(* CODESYS project Initial_Program.project
   Version: 0.0.0.0
   Title: Initial_Program
   Author: MYBOOK

Project tree, tasks and I/O mapping:
  Skripsi_Yosef : TM262L10MESE8T, Schneider Electric, order no. TM262L10MESE8T, version 5.0.4.83
      settings: Enable OPC-UA Server = True; BinaryFileSize = 1168; Dhcps Host 0.Client Device Name = 'DEVICE_1'; Dhcps Host 0.Client IP Address = [192, 168, 3, 200]; Dhcps Host 0.Network Mask = [255, 255, 255, 0]; Dhcps Host 0.Default Gateway = [192, 168, 3, 254]; Dhcps Host 1.Client Device Name = 'DEVICE_2'; Dhcps Host 1.Client IP Address = [192, 168, 3, 100]; Dhcps Host 1.Network Mask = [255, 255, 255, 0]; Dhcps Host 1.Default Gateway = [192, 168, 3, 254]; Dhcps Host 2.Client Device Name = 'DEVICE_3'; Dhcps Host 2.Client IP Address = [192, 168, 3, 201]; Dhcps Host 2.Network Mask = [255, 255, 255, 0]; Dhcps Host 2.Default Gateway = [192, 168, 3, 254]; Dhcps Host 3.Client Device Name = 'DEVICE_4'; Dhcps Host 3.Client IP Address = [192, 168, 3, 101]; Dhcps Host 3.Network Mask = [255, 255, 255, 0]; Dhcps Host 3.Default Gateway = [192, 168, 3, 254]; Dhcps Host 4.Client Device Name = 'DEVICE_5'; Dhcps Host 4.Client IP Address = [192, 168, 3, 203]; Dhcps Host 4.Network Mask = [255, 255, 255, 0]; Dhcps Host 4.Default Gateway = [192, 168, 3, 254]; Dhcps Host 5.Client Device Name = 'DEVICE_6'; Dhcps Host 5.Client IP Address = [192, 168, 3, 202]; Dhcps Host 5.Network Mask = [255, 255, 255, 0]; Dhcps Host 5.Default Gateway = [192, 168, 3, 254]; InterfaceUsedByDhcpSize = 4; InterfaceUsedByDhcp = [192,168,3,254]
    application Application
      task MAST (cyclic, interval 10 ms, priority 15, watchdog 50 ms x 1) calls SR_Main
      program SR_Main [LD]
      global variables GVL
      program POU [SFC]
    Machine Assistant
    Message Logger
    COM_Bus : COM Bus - TMS, Schneider Electric, version 5.0.4.83
    Ethernet_1 : ETH1, Schneider Electric, version 5.0.4.83
        settings: DeviceName = 'M262'; WebServer = FALSE; FTP Server = TRUE; SoMachine Protocol = FALSE; Modbus Server = FALSE; NetManage Protocol = FALSE; SNMP protocol = FALSE; WebVisu protocol = FALSE; DHCP Server Active = TRUE; Secured Web Server = TRUE; Remote Connection = FALSE
    Ethernet_2 : ETH2, Schneider Electric, version 5.0.4.83
        settings: IPAddress = [192, 168, 3, 254]; SubnetMask = [255, 255, 255, 0]; GatewayAddress = [192, 168, 3, 1]; DeviceName = 'M262_PLC'; WebServer = TRUE; FTP Server = FALSE; SoMachine Protocol = TRUE; Modbus Server = TRUE; NetManage Protocol = TRUE; SNMP protocol = TRUE; WebVisu protocol = TRUE; DHCP Server Active = TRUE; Secured Web Server = TRUE; Remote Connection = TRUE
      Modbus_TCP_IO_Scanner : Modbus TCP IO Scanner, Schneider Electric, version 1.0.0.12
          unmapped channels: Global Status, Healthbit 0, Healthbit 1, Healthbit 2, Healthbit 3
        OT_Sensor_Temp_Humid : Generic Modbus TCP Slave, Schneider Electric, version 1.0.2.21
            settings: DeviceNumber = 512; Object Input1 = [128, 2, 21233664, 0]; Unit-ID = 248; IPAddress = [192, 168, 3, 200]; GatewayAddress = [192, 168, 3, 254]; DeviceName = 'DEVICE_1'; Channel 0.Channel ID = 0; Channel 0.Unit-ID = 1; Channel 0.Repetition Rate = 100; Channel 0.Function Code = 3; Channel 0.Read Offset = 16#0000; Channel 0.Read Length = 2; Channel 0.Write Offset = 0; Channel 0.Write Length = 0
            unmapped channels: Channel 0, Channel 0
        AHU_Act_Remote_AC : Generic Modbus TCP Slave, Schneider Electric, version 1.0.2.21
            settings: DeviceNumber = 513; Object Output1 = [131, 2, 25428068, 1]; Unit-ID = 248; IPAddress = [192, 168, 3, 100]; GatewayAddress = [192, 168, 3, 254]; DeviceName = 'DEVICE_2'; Channel 1.Channel ID = 1; Channel 1.Unit-ID = 255; Channel 1.Repetition Rate = 100; Channel 1.Function Code = 16; Channel 1.Read Offset = 0; Channel 1.Read Length = 0; Channel 1.Write Offset = 16#0064; Channel 1.Write Length = 2
            unmapped channels: Channel 1, Channel 1
        OT_Sensor_Press_Temp : Generic Modbus TCP Slave, Schneider Electric, version 1.0.2.21
            settings: DeviceNumber = 514; Object Input1 = [132, 2, 21233764, 2]; Unit-ID = 248; IPAddress = [192, 168, 3, 201]; GatewayAddress = [192, 168, 3, 254]; DeviceName = 'DEVICE_3'; Channel 1.Channel ID = 2; Channel 1.Unit-ID = 255; Channel 1.Repetition Rate = 100; Channel 1.Function Code = 3; Channel 1.Read Offset = 16#0064; Channel 1.Read Length = 2; Channel 1.Write Offset = 0; Channel 1.Write Length = 0
            unmapped channels: Channel 1, Channel 1
        AHU_Act_Motor_Exhaust : Generic Modbus TCP Slave, Schneider Electric, version 1.0.2.21
            settings: DeviceNumber = 515; Object Output1 = [135, 8, 25427968, 3]; Unit-ID = 248; IPAddress = [192, 168, 3, 101]; GatewayAddress = [192, 168, 3, 254]; DeviceName = 'DEVICE_4'; Channel 3.Channel ID = 3; Channel 3.Unit-ID = 1; Channel 3.Repetition Rate = 100; Channel 3.Function Code = 16; Channel 3.Read Offset = 0; Channel 3.Read Length = 0; Channel 3.Write Offset = 16#0000; Channel 3.Write Length = 8
            unmapped channels: Channel 3, Channel 3, Channel 3, Channel 3, Channel 3, Channel 3, Channel 3, Channel 3
        AHU_Sensor_Temp_Humid_Pressure : Generic Modbus TCP Slave, Schneider Electric, version 1.0.2.21
            settings: DeviceNumber = 516; Object Input1 = [136, 4, 21233764, 4]; Unit-ID = 248; IPAddress = [192, 168, 3, 203]; GatewayAddress = [192, 168, 3, 254]; DeviceName = 'DEVICE_5'; Channel 4.Channel ID = 4; Channel 4.Unit-ID = 255; Channel 4.Repetition Rate = 20; Channel 4.Function Code = 3; Channel 4.Read Offset = 16#0064; Channel 4.Read Length = 4; Channel 4.Write Offset = 0; Channel 4.Write Length = 0
            unmapped channels: Channel 4, Channel 4, Channel 4, Channel 4
        Outdoor_Sensor_Press_temp : Generic Modbus TCP Slave, Schneider Electric, version 1.0.2.21
            settings: DeviceNumber = 517; Object Input1 = [138, 2, 21233764, 5]; Unit-ID = 248; IPAddress = [192, 168, 3, 202]; GatewayAddress = [192, 168, 3, 254]; DeviceName = 'DEVICE_6'; Channel 5.Channel ID = 5; Channel 5.Unit-ID = 255; Channel 5.Repetition Rate = 20; Channel 5.Function Code = 3; Channel 5.Read Offset = 16#0064; Channel 5.Read Length = 2; Channel 5.Write Offset = 0; Channel 5.Write Length = 0
            unmapped channels: Channel 5, Channel 5
    Serial_Line : Serial line, Schneider Electric, version 5.0.4.83
      Machine_Expert_Network_Manager : Machine Expert-Network Manager, Schneider Electric, version 4.0.0.3
    DI : Digital Inputs, Schneider Electric, version 5.0.4.83
        input  ibDI_IB0 : BYTE  // IB0
        input  ibDI_IB1 : BYTE  // IB1
    DQ : Digital Outputs, Schneider Electric, version 5.0.4.83
        unmapped channels: QB0, QB1
    IO_Bus : IO bus - TM3, Schneider Electric, version 5.0.4.83
  FdtConnections : FDT Connections, Schneider Electric, version 1.0.0.2
  Project Information/
    function GetCompany [ST]
    function GetTitle [ST]
    function GetVersion [ST]
    function GetTextProperty [ST]
    function GetTextProperty2 [ST]
    function GetNumberProperty [ST]
    function GetBooleanProperty [ST]
    function GetVersionProperty [ST]
*)

// Skripsi_Yosef/Application/GVL
{attribute 'qualified_only'}
VAR_GLOBAL
	
END_VAR

// Skripsi_Yosef/Application/SR_Main
PROGRAM SR_Main
VAR
	AC_StatusHMI AT %MX6.0: BOOL := FALSE;
	OT_Temp AT %MW0: WORD;
	OT_Humid AT %MW1: WORD;
	OT_Pressure AT %MW2: WORD;
	AC_Status AT %MW4: WORD;
	AC_Temp AT %MW5: WORD := 24;
	AC_TempUp AT %MX12.0: BOOL;
	AC_TempDown AT %MX12.1: BOOL;
	AC_TempRST AT %MX12.2: BOOL;
	AHU_Temp AT %MW7: WORD;
	AHU_Humid AT %MW8: WORD;
	AHU_Press AT %MW9: WORD;
	AHU_FanOverride AT %MX20.0: BOOL;
	HMI_FANSpeed1 AT %MW11: WORD;
	HMI_FANSpeed2 AT %MW12: WORD;
	HMI_FANSpeed3 AT %MW13: WORD;
	HMI_FANSpeed4 AT %MW14: WORD;
	OT_TempSP AT %MW15: WORD := 230;
	OT_TempSPUp AT %MX32.0: BOOL;
	OT_TempSPDown AT %MX32.1: BOOL;
	OT_BuildingTemp AT %MW17: WORD;
	Outdoor_Press AT %MW18: WORD;
	Outdoor_Temp AT %MW19: WORD;
	z2e_CtlSig: REAL;
	e_CtlSig: REAL;
	u_CtlSig: REAL;
	a1: REAL;
	b1: REAL;
	b2: REAL;
	b3: REAL;
	b4: REAL;
	b5: REAL;
	c1: REAL;
	c2: REAL;
	c3: REAL;
	f1: REAL;
	f2: REAL;
	Qac_joule: REAL;
	k1: REAL := 2;
	k2: REAL := 2;
	kmz: REAL := 343;
	kom: REAL := 34.3;
	Cm: REAL := 2301;
	rho_a: REAL := 1.18;
	Vc: REAL := 4;
	Vz: REAL := 0.576;
	Qac_btu: REAL := 5000;
	Cpa: REAL := 700;
	PWM_FanSpeed1 AT %MW20: WORD;
	PWM_FanSpeed2 AT %MW21: WORD;
	PWM_FanSpeed3 AT %MW22: WORD;
	PWM_FanSpeed4 AT %MW23: WORD;
	ErrorRatio: REAL;
END_VAR
VAR // added by the converter: edge detectors and wires of the graphical bodies
    _rt1, _rt2, _rt3, _rt4 : R_TRIG;
    _w1, _w2, _w3, _w4, _w5 : BOOL;
END_VAR

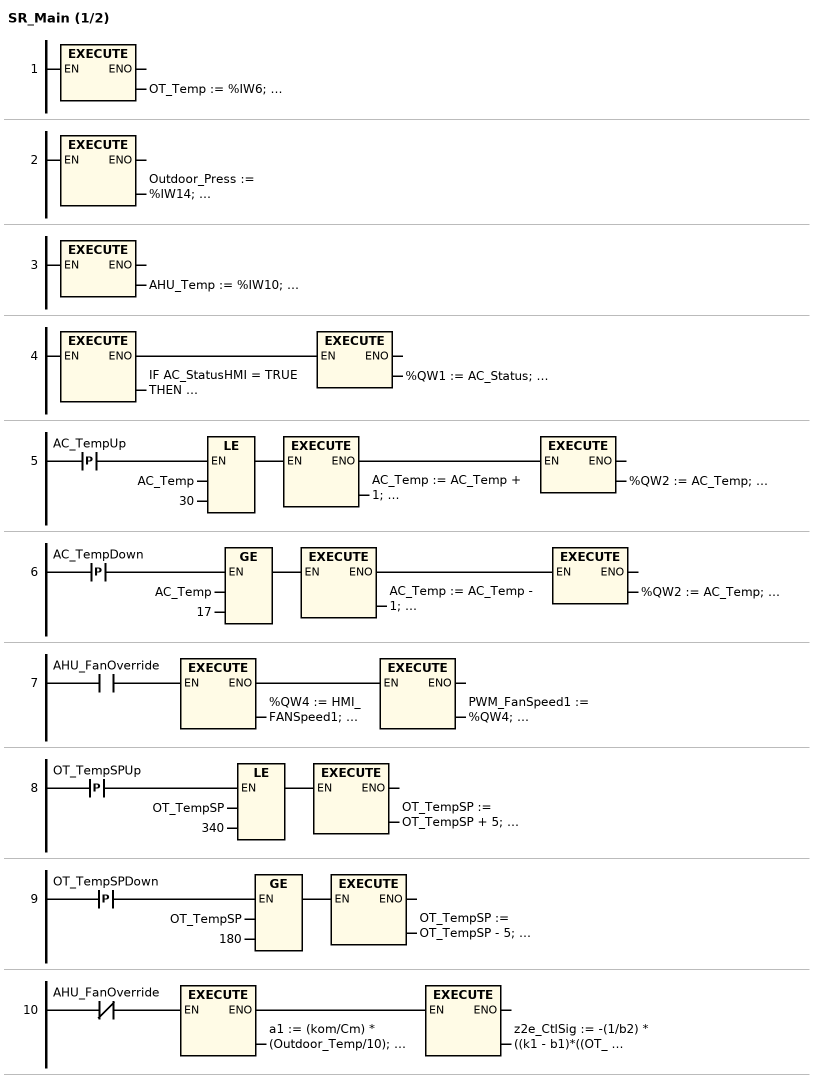
// NETWORK 1
OT_Temp := %IW6;
OT_Humid := %IW7;
OT_Pressure := %IW8;
OT_BuildingTemp := %IW9;

// NETWORK 2
Outdoor_Press := %IW14;
Outdoor_Temp := %IW15;

// NETWORK 3
AHU_Temp := %IW10;
AHU_Humid := %IW11;
AHU_Press := %IW13;

// NETWORK 4
IF AC_StatusHMI = TRUE THEN
	AC_Status := 1;
END_IF

IF AC_StatusHMI = FALSE THEN
	AC_Status := 0;
END_IF
%QW1 := AC_Status;

// NETWORK 5
_rt1(CLK := AC_TempUp);
_w1 := _rt1.Q AND AC_Temp <= 30;
IF _w1 THEN AC_Temp := AC_Temp + 1; END_IF
IF _w1 THEN %QW2 := AC_Temp; END_IF

// NETWORK 6
_rt2(CLK := AC_TempDown);
_w2 := _rt2.Q AND AC_Temp >= 17;
IF _w2 THEN AC_Temp := AC_Temp - 1; END_IF
IF _w2 THEN %QW2 := AC_Temp; END_IF

// NETWORK 7
_w3 := AHU_FanOverride;
IF _w3 THEN
    %QW4 := HMI_FANSpeed1;
    %QW6 := HMI_FANSpeed2;
    %QW8 := HMI_FANSpeed3;
    %QW10 := HMI_FANSpeed4;
END_IF
IF _w3 THEN
    PWM_FanSpeed1 := %QW4;
    PWM_FanSpeed2 := %QW6;
    PWM_FanSpeed3 := %QW8;
    PWM_FanSpeed4 := %QW10;
END_IF

// NETWORK 8
_rt3(CLK := OT_TempSPUp);
IF _rt3.Q AND OT_TempSP <= 340 THEN OT_TempSP := OT_TempSP + 5; END_IF

// NETWORK 9
_rt4(CLK := OT_TempSPDown);
IF _rt4.Q AND OT_TempSP >= 180 THEN OT_TempSP := OT_TempSP - 5; END_IF

// NETWORK 10
_w4 := NOT AHU_FanOverride;
IF _w4 THEN
    a1 := (kom/Cm) * (Outdoor_Temp/10);
    b1 := (kmz + kom)/Cm;
    b2 := kmz/Cm;
    b3 := kmz/(rho_a * Cpa * Vz);
    b4 := 1/Vz;
    b5 := 1/Vc;
    c1 := b3 - ((k1 - b3)*(k1 - b1))/b2;
    c2 := k1 - b1 - b3;
    c3 := (k1 - b1)/b2;
    f1 := -(a1/b2) + b1*(OT_TempSP/10)/b2;
    f2 := ((b3 * a1)/b2) + (b3 * (b2 - b1)/b2)*(OT_TempSP/10);
END_IF
IF _w4 THEN
    z2e_CtlSig := -(1/b2) * ((k1 - b1)*((OT_BuildingTemp-OT_TempSP)/10) + a1 + (b2 - b1)*(OT_TempSP/10));
    
    e_CtlSig :=  (OT_Temp - OT_TempSP)/10 - z2e_CtlSig;
    
    u_CtlSig := ((c1 + b2)*((OT_BuildingTemp - OT_TempSP)/10)+(c2 + k2)*e_CtlSig + f2)/(b4 * (e_CtlSig - c3*((OT_Temp - OT_TempSP)/10) - (AHU_Temp/10) + f1));
END_IF

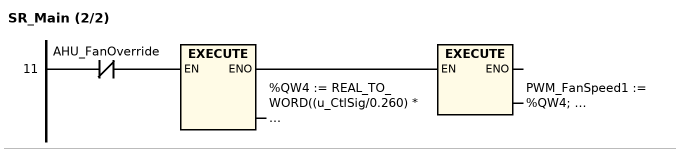
// NETWORK 11
_w5 := NOT AHU_FanOverride;
IF _w5 THEN
    %QW4 := REAL_TO_WORD((u_CtlSig/0.260) * 100);
    IF %QW4 >= 100 THEN
    	%QW4 := 100;
    ELSIF %QW4 <= 20 THEN
    	%QW4 := 20;
    END_IF
    %QW6 := REAL_TO_WORD((u_CtlSig/0.260) * 100);
    IF %QW6 >= 100 THEN
    	%QW6 := 100;
    ELSIF %QW6 <= 20 THEN
    	%QW6 := 20;
    END_IF
    %QW8 := REAL_TO_WORD((u_CtlSig/0.260) * 100);
    IF %QW8 >= 100 THEN
    	%QW8 := 100;
    ELSIF %QW8 <= 20 THEN
    	%QW8 := 20;
    END_IF
    %QW10 := 100;
    
    ErrorRatio := OT_Temp - OT_TempSP;
    
    IF ErrorRatio <= 0 THEN
    	%QW4 := 40;
    	%QW6 := 40;
    	%QW8 := 40;
    END_IF
END_IF
IF _w5 THEN
    PWM_FanSpeed1 := %QW4;
    PWM_FanSpeed2 := %QW6;
    PWM_FanSpeed3 := %QW8;
    PWM_FanSpeed4 := %QW10;
END_IF

END_PROGRAM

// Project Information/GetCompany
// This function has been automatically generated from the project information.
{attribute 'signature_flag' := '1073741824'}
{attribute 'register_in_runtime'}
FUNCTION GetCompany : WSTRING
VAR_INPUT
	
END_VAR

GetCompany := "";

END_FUNCTION

// Project Information/GetTitle
// This function has been automatically generated from the project information.
{attribute 'signature_flag' := '1073741824'}
{attribute 'register_in_runtime'}
FUNCTION GetTitle : WSTRING
VAR_INPUT
	
END_VAR

GetTitle := "Initial_Program";

END_FUNCTION

// Project Information/GetVersion
// This function has been automatically generated from the project information.
{attribute 'signature_flag' := '1073741824'}
{attribute 'register_in_runtime'}
FUNCTION GetVersion : VERSION
VAR_INPUT
	
END_VAR

GetVersion.uiMajor := 0;
GetVersion.uiMinor := 0;
GetVersion.uiServicePack := 0;
GetVersion.uiPatch := 0;

END_FUNCTION

// Project Information/GetTextProperty
// This function has been automatically generated from the project information.
{attribute 'signature_flag' := '1073741824'}
{attribute 'register_in_runtime'}
FUNCTION GetTextProperty : WSTRING
VAR_INPUT
	stKey: WSTRING;
END_VAR

IF stKey = "Author" THEN
	GetTextProperty := "MYBOOK";
ELSIF stKey = "Company" THEN
	GetTextProperty := "";
ELSIF stKey = "Description" THEN
	GetTextProperty := "";
ELSIF stKey = "Project" THEN
	GetTextProperty := "Initial_Program";
ELSIF stKey = "Title" THEN
	GetTextProperty := "Initial_Program";
ELSE
	GetTextProperty := "";
END_IF

END_FUNCTION

// Project Information/GetTextProperty2
// This function has been automatically generated from the project information.
{attribute 'signature_flag' := '1073741824'}
{attribute 'register_in_runtime'}
FUNCTION GetTextProperty2 : POINTER TO WSTRING
VAR_INPUT
	stKey: WSTRING;
END_VAR

IF stKey = "Author" THEN
	GetTextProperty2 := ADR("MYBOOK");
ELSIF stKey = "Company" THEN
	GetTextProperty2 := ADR("");
ELSIF stKey = "Description" THEN
	GetTextProperty2 := ADR("");
ELSIF stKey = "Project" THEN
	GetTextProperty2 := ADR("Initial_Program");
ELSIF stKey = "Title" THEN
	GetTextProperty2 := ADR("Initial_Program");
ELSE
	GetTextProperty2 := ADR("");
END_IF

END_FUNCTION

// Project Information/GetNumberProperty
// This function has been automatically generated from the project information.
{attribute 'signature_flag' := '1073741824'}
{attribute 'register_in_runtime'}
FUNCTION GetNumberProperty : DINT
VAR_INPUT
	stKey: WSTRING;
END_VAR

GetNumberProperty := 0;

END_FUNCTION

// Project Information/GetBooleanProperty
// This function has been automatically generated from the project information.
{attribute 'signature_flag' := '1073741824'}
{attribute 'register_in_runtime'}
FUNCTION GetBooleanProperty : BOOL
VAR_INPUT
	stKey: WSTRING;
END_VAR

GetBooleanProperty := FALSE;

END_FUNCTION

// Project Information/GetVersionProperty
// This function has been automatically generated from the project information.
{attribute 'signature_flag' := '1073741824'}
{attribute 'register_in_runtime'}
FUNCTION GetVersionProperty : VERSION
VAR_INPUT
	stKey: WSTRING;
END_VAR

IF stKey = "Version" THEN
	GetVersionProperty.uiMajor := 0;
	GetVersionProperty.uiMinor := 0;
	GetVersionProperty.uiServicePack := 0;
	GetVersionProperty.uiPatch := 0;
ELSE
	GetVersionProperty.uiMajor := 0;
	GetVersionProperty.uiMinor := 0;
	GetVersionProperty.uiServicePack := 0;
	GetVersionProperty.uiPatch := 0;
END_IF

END_FUNCTION

// Skripsi_Yosef/Application/POU
PROGRAM POU
VAR
END_VAR

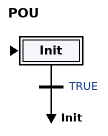
INITIAL_STEP Init:
END_STEP
TRANSITION FROM Init TO Init
    := TRUE;
END_TRANSITION

END_PROGRAM
